FUNCTION_BLOCK FB_SecondaryControlSinus
VAR_INPUT
	ThetaRef 			: LREAL; // Kul
	fPosition 			: LREAL; 
	
END_VAR
VAR_OUTPUT
END_VAR
VAR
END_VAR

END_FUNCTION_BLOCK

(* stored: Version 1.1.0.1
   POU FB_SecondaryControlSinus: Id {4e1fc59f-b966-4ece-96fa-c350a8c20e41}, SpecialFunc None *)
